{attribute 'qualified_only'}
VAR_GLOBAL
	{attribute 'OPC.UA.DA' := '1'}
	{attribute 'OPC.UA.DA.Access' := '1'}
	{attribute 'init_namespace'} 
	Name : STRING(255);	
END_VAR

(* stored: Version 1.1.0.1
   GVL CurrentNamespace: Id {a4f4d352-e135-49fe-9d76-2fb59cdf58f2} *)
